Fanuc KAREL source: compact_preamble.KL

PROGRAM KB00044
%NOLOCKGROUP
%ENVIRONMENT TPE
VAR
P1 : STRING[80];P2 : STRING[80]
P3 : FILE
P4:BOOLEAN
P5:INTEGER
P6:INTEGER
BEGIN
P1='A'
P2='A'
P4=TRUE
P5=1
P6=1
COMPARE_FILE(P1,P2,P3,P4,P5,P6)
END KB00044
